FUNCTION_BLOCK Derivative
VAR_INPUT
	rValue:LREAL;			(*Valor a ser derivado*)
	rPastTime:LREAL;		(*tempo decorrido em ms*)
END_VAR
VAR_OUTPUT
	rDerivative:LREAL;		(*valor derivado*)
END_VAR
VAR
	rOldValue: LREAL;
END_VAR

IF rPastTime>0 THEN
	rDerivative:=(rValue-rOldValue)/rPastTime;
ELSE
	rDerivative:=0;
END_IF
rOldValue:=rValue;

END_FUNCTION_BLOCK

(* stored: Version 1.1.0.1, ProductVersion 3.1.4024.12
   POU Derivative: Id {9c2d971f-073e-44dd-991f-64c8def17c78}, SpecialFunc None *)
